KUKA KRL data list: mes_info.dat

&ACCESS RVP3
&REL 7882
&PARAM EDITMASK = *
&PARAM TEMPLATE = C:\KRC\Roboter\Template\vorgabe
&PARAM DISKPATH = KRC:\R1\Program\HG
DEFDAT  MES_INFO PUBLIC

DECL DATE Robot_Run_Time

GLOBAL INT T1_Time=0
GLOBAL INT Aut_Time=0

GLOBAL INT Work_A_Run_Cycle_Time=0
GLOBAL INT Work_A_Run_All_Time=0
GLOBAL INT Work_B_Run_Cycle_Time=0
GLOBAL INT Work_B_Run_All_Time=0
GLOBAL INT Work_C_Run_Cycle_Time=0
GLOBAL INT Work_C_Run_All_Time=0
GLOBAL INT Work_D_Run_Cycle_Time=0
GLOBAL INT Work_D_Run_All_Time=0

GLOBAL BOOL WORK_A_State=FALSE
GLOBAL BOOL WORK_B_State=FALSE
GLOBAL BOOL WORK_C_State=FALSE
GLOBAL BOOL WORK_D_State=FALSE

GLOBAL INT Socket_TimeOut=50

GLOBAL INT Work_A_Run_Nunber=0
GLOBAL INT Work_B_Run_Nunber=0
GLOBAL INT Work_C_Run_Nunber=0
GLOBAL INT Work_D_Run_Nunber=0
GLOBAL INT Work_All_Run_Nunber=0
GLOBAL CHAR DATAPATH_NAME[1024]



DECL BOOL _Work_A_Stat=FALSE
DECL BOOL _Work_B_Stat=FALSE
DECL BOOL _Work_C_Stat=FALSE
DECL BOOL _Work_D_Stat=FALSE
DECL BOOL _EKRL_Connect_Stat=FALSE
DECL BOOL _EKRL_Send_Stat=FALSE

DECL BOOL _EKRL_Server_Connt_Stat=FALSE

GLOBAL CONST CHAR Robot_Process_Name[1024]
Robot_Process_Name[]="Spot_Surround_1"


ENDDAT
